// Mitsubishi GX Works2 project: 시퀀스 회로 (무한 반복)   PLC: Q03UDV

PROGRAM MAIN
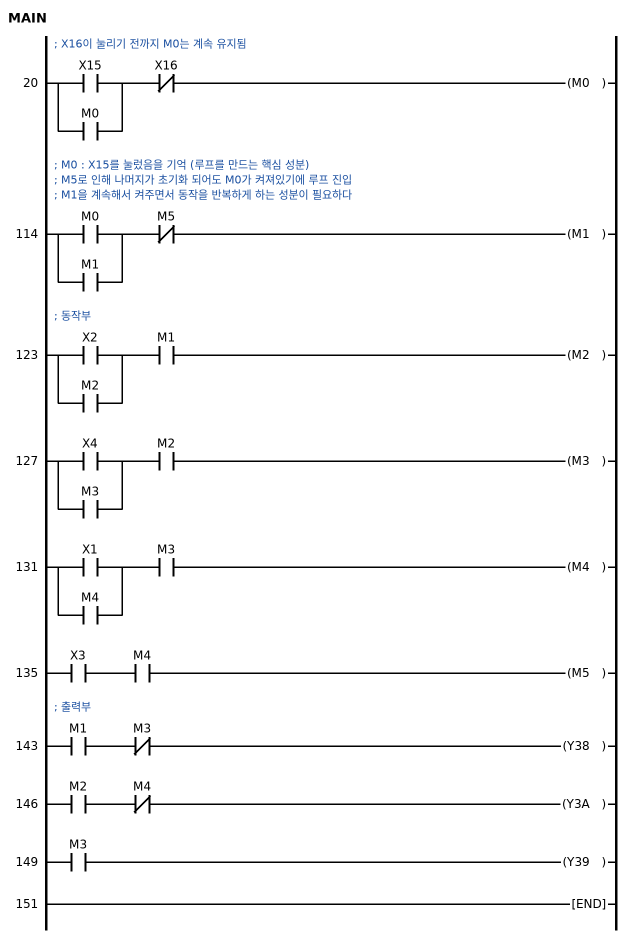
; X16이 눌리기 전까지 M0는 계속 유지됨
20    LD      X15
      OR      M0
      ANI     X16
      OUT     M0
; M0 : X15를 눌렀음을 기억 (루프를 만드는 핵심 성분)
; M5로 인해 나머지가 초기화 되어도 M0가 켜져있기에 루프 진입
; M1을 계속해서 켜주면서 동작을 반복하게 하는 성분이 필요하다
114   LD      M0
      OR      M1
      ANI     M5
      OUT     M1
; 동작부
123   LD      X2
      OR      M2
      AND     M1
      OUT     M2
127   LD      X4
      OR      M3
      AND     M2
      OUT     M3
131   LD      X1
      OR      M4
      AND     M3
      OUT     M4
135   LD      X3
      AND     M4
      OUT     M5
; 출력부
143   LD      M1
      ANI     M3
      OUT     Y38
146   LD      M2
      ANI     M4
      OUT     Y3A
149   LD      M3
      OUT     Y39
151   END
END_PROGRAM
